TYPE HMIWorkpieceInterface :
STRUCT
	WorkpieceSettingLines	:	ARRAY[1..3] of HMISettingLineInterface;	
END_STRUCT
END_TYPE

(* stored: Version 1.1.0.1
   DUT HMIWorkpieceInterface: Id {73d13c24-ca17-41e6-818b-9b7d2b7d0190} *)
